
FUNCTION CB_sint_to_dint : DINT

TITLE = ' Convert an integer into a Dint '
VERSION : '1.0'
AUTHOR  : CB
NAME    : sinToDin
FAMILY  : TNI

VAR_INPUT
    IN : INT;
END_VAR

BEGIN

CB_sint_to_dint := IN;

END_FUNCTION
